KUKA KRL program: RoboSyncStepper.src, RoboSyncStepper.dat

--- RoboSyncStepper.src ---
&ACCESS RVO3
&REL 16
&PARAM DISKPATH = KRC:\R1\TP\CNCRobotics\CEAD
DEF RoboSyncStepper( )
;************************************************
;     NextState Automation Ltd
;     www.nextstateautomation.co.uk
;************************************************
;     Contact: helpdesk@nextstateautomation.co.uk
;     Date: 14/09/26
;     Version: 0.1.1
;     Module : RoboSyncStepper
;     Purpose: Stepper drive commands and parameters for the RoboSync Hub
;************************************************
END

GLOBAL DEF SetStepperParam(fi_param:IN, fi_nVal:IN)
;------------------------------------------------
; Name    : SetStepperParam
; Purpose : Write one stepper drive parameter
; Params  : fi_param   (IN) ENUM_STEPPER_PARAM : parameter to write
;           fi_nVal    (IN) INT                : value, in the drive units
; Returns : -
; Notes   : Takes control from the SPS while writing. Units (hub guide):
;           current 0.01 A, pulse/rev = ppr/2, jog speed 0.25 RPM (signed),
;           accel/decel 10 RPM/s, distance pulses.
;           Robot interpreter only (WAIT)
;------------------------------------------------
DECL ENUM_STEPPER_PARAM fi_param
DECL INT fi_nVal
BOOL _bFlag

_bFlag = bspsControl
bSpsControl = FALSE
WAIT FOR bProcessing==FALSE

SWITCH fi_param

   CASE #CURRENT
      stepper_Current = fi_nVal
   CASE #IDLE_CURRENT
      stepper_idleCurrent = fi_nVal
   CASE #PULSE_PER_REV
      stepper_pulsePerRev = fi_nVal
   CASE #JOG_SPEED
      stepper_jogSpeed = ToUnsigned16(fi_nVal)
   CASE #JOG_ACCEL
     stepper_jogAccel = fi_nVal
   CASE #JOG_DECEL
     stepper_jogDecel = fi_nVal
   CASE #SPEED
      stepper_speed = fi_nVal
   CASE #ACCEL
      stepper_Accel = fi_nVal
   CASE #DECEL
      stepper_Decel = fi_nVal
   CASE #DISTANCE
      stepper_Dist = fi_nVal
   CASE #SET_POSITION ;This might need to be performed in a single write
      stepper_OpCode2 = 0
      stepper_OpCode2Param = fi_nVal
      stepper_OpCode2 = SET_POSITION

ENDSWITCH

bspsControl = _bFlag
END

GLOBAL DEF StepperOpcode(fi_nVal:IN)
;------------------------------------------------
; Name    : StepperOpcode
; Purpose : Write a command to the stepper opcode register
; Params  : fi_nVal    (IN) INT : opcode, e.g. ENABLE_DRIVE
; Returns : -
; Notes   : Leave time for the drive to act before writing the next
;           opcode, see nStepperCmdDelay
;------------------------------------------------
DECL INT fi_nVal

   stepper_OpCode = fi_nVal

END

GLOBAL DEF StartJog( fi_nVal:IN )
;------------------------------------------------
; Name    : StartJog
; Purpose : Reset alarms, enable the drive and start jogging manually,
;           e.g. to purge or load filament
; Params  : fi_nVal    (IN) INT : jog speed, 0.25 RPM units, negative reverses
; Returns : -
; Notes   : Do not use while the SPS state machine controls the stepper.
;           Robot interpreter only (WAIT)
;------------------------------------------------
DECL INT fi_nVal

;Each opcode needs time to reach the drive before the next is written
StepperOpcode(RESET_ALARM_CODE)
WAIT SEC nStepperCmdDelay/1000.0

SetStepperParam(#JOG_ACCEL,nJogAccel)
SetStepperParam(#JOG_DECEL,nJogDecel)
StepperOpcode(ENABLE_DRIVE)
WAIT SEC nStepperCmdDelay/1000.0

SetStepperParam(#JOG_SPEED,fi_nVal)
WAIT SEC nStepperStartDelay/1000.0
StepperOpcode(COMMENCE_JOGGING)

END

GLOBAL DEF StopJog( )
;------------------------------------------------
; Name    : StopJog
; Purpose : Stop manual jogging
; Params  : -
; Returns : -
;------------------------------------------------

StepperOpcode(STOP_JOGGING)
END

GLOBAL DEFFCT BOOL StepperError()
;------------------------------------------------
; Name    : StepperError
; Purpose : Check the stepper drive alarm code
; Params  : -
; Returns : BOOL, TRUE if any alarm bit is set
;------------------------------------------------

RETURN stepper_alarm<>0

 ;stepper_positionLimit
; stepper_ccwLimit
 ;stepper_cwLimit
; stepper_overTemperature
; stepper_interalVoltage
 ;stepper_overVoltage
; stepper_underVoltage
; stepper_overCurrent

 ;stepper_openMotorWinding
 ;stepper_encoderError
 ;stepper_commsError
 ;stepper_flashError
 ;stepper_NoMove
 ;stepper_AlarmSpare1
 ;stepper_blankQSegment
 ;stepper_AlarmSpare2
ENDFCT

GLOBAL DEFFCT INT ToUnsigned16(fi_nVal:IN)
;------------------------------------------------
; Name    : ToUnsigned16
; Purpose : Encode a signed value as 16 bit two's complement for an
;           output word
; Params  : fi_nVal    (IN) INT : -32768..32767
; Returns : INT, 0..65535
;------------------------------------------------
;Two's complement encoding of a signed value for a 16 bit output
DECL INT fi_nVal

IF fi_nVal < 0 THEN
   RETURN 65536 + fi_nVal
ENDIF
RETURN fi_nVal
ENDFCT

GLOBAL DEFFCT INT Truncate16(n:IN)
;------------------------------------------------
; Name    : Truncate16
; Purpose : Keep only the low 16 bits of an INT
; Params  : n          (IN) INT
; Returns : INT
; Notes   : Unused and untested, ToUnsigned16 is used instead
;------------------------------------------------

DECL INT ofs
DECL INT n, nOut
DECL CHAR buf[4]


ofs=0
cast_to(buf[],ofs,n)

buf[3] = 0
buf[4] = 0

ofs=0
cast_from(buf[],ofs,nOut)

return nOut
ENDFCT

--- RoboSyncStepper.dat ---
&ACCESS RVO3
&REL 16
&PARAM DISKPATH = KRC:\R1\TP\CNCRobotics\CEAD
DEFDAT  RoboSyncStepper PUBLIC
;************************************************
;     NextState Automation Ltd
;     www.nextstateautomation.co.uk
;************************************************
;     Contact: helpdesk@nextstate.co.uk
;     Date: 14/09/26
;     Version: 0.1.1
;************************************************

GLOBAL CONST INT RESET_ALARM_CODE=186
GLOBAL CONST INT ENABLE_DRIVE=159
GLOBAL CONST INT DISABLE_DRIVE=158
GLOBAL CONST INT COMMENCE_JOGGING=150
GLOBAL CONST INT STOP_JOGGING=216
GLOBAL CONST INT MOVE_RELATIVE_DISTANCE=102
GLOBAL CONST INT MOVE_ABSOLUTE_DISTANCE=103
GLOBAL CONST INT FAST_STOP_MOVE=225
GLOBAL CONST INT STOP_MOVE=226
GLOBAL CONST INT SET_POSITION = 165

GLOBAL ENUM ENUM_STEPPER_PARAM CURRENT,IDLE_CURRENT,PULSE_PER_REV,JOG_SPEED,JOG_ACCEL,JOG_DECEL,SPEED,ACCEL,DECEL,DISTANCE,SET_POSITION

ENDDAT
